{attribute 'qualified_only'}
VAR_GLOBAL
END_VAR

(* stored: Version 1.1.0.1, ProductVersion 3.1.4024.16
   GVL IO1: Id {7c657149-8db4-4c36-a944-7ccff1440f5d} *)
